// TwinCAT 3 PLC project PLC1
// ProgramVersion: 3.1.4024.0
// libraries:
//   Tc2_Standard, * (Beckhoff Automation GmbH)
//   Tc2_System, * (Beckhoff Automation GmbH)
//   Tc3_Module, * (Beckhoff Automation GmbH)
// project tree:
//   GVLs/ GVL.TcGVL
//   / PlcTask.TcTTO
//   POUs/ MAIN.TcPOU, P001_Counter1.TcPOU, P002_TestAnother.TcPOU
// real-time tasks:
//   TASK PlcTask: cycle T#10ms, priority 20, ADS port 350
// I/O:
//   DEVICE Device 1 (EtherCAT), AmsNetId 192.168.196.219.2.1
//     Term 1 (EK1100) [EK1100 EtherCAT Coupler (2A E-Bus)]
//       Term 2 (EL1809) [EL1809 16Ch. Dig. Input 24V, 3ms]
//       Term 3 (EL1809) [EL1809 16Ch. Dig. Input 24V, 3ms] (disabled)
//       Term 4 (EL2809) [EL2809 16Ch. Dig. Output 24V, 0.5A] (disabled)
//       Term 5 (EL2809) [EL2809 16Ch. Dig. Output 24V, 0.5A] (disabled)

CONFIGURATION PLC1
    RESOURCE PLC ON TwinCAT3
        TASK PlcTask(INTERVAL := T#10ms, PRIORITY := 20);
        PROGRAM MAIN WITH PlcTask : MAIN;
    END_RESOURCE
END_CONFIGURATION

// ---- GVLs/GVL.TcGVL
{attribute 'qualified_only'}
VAR_GLOBAL
	iInt	: UDINT;
END_VAR

// ---- POUs/MAIN.TcPOU
PROGRAM MAIN
VAR
	bInit: BOOL;
	Test123: INT;
END_VAR

IF NOT bInit THEN
	bInit:=TRUE;
END_IF

P001_Counter1();
Test123:=2;

END_PROGRAM

// ---- POUs/P001_Counter1.TcPOU
PROGRAM P001_Counter1
VAR
	count: INT;
END_VAR

count:=count+1;

END_PROGRAM

// ---- POUs/P002_TestAnother.TcPOU
PROGRAM P002_TestAnother
VAR
	Count: INT;
	bInit: BOOL;
END_VAR

Count:=Count+2;
IF NOT bInit THEN
	bInit:=TRUE;
END_IF

END_PROGRAM
